PROGRAM Clamp_and_cut
VAR
	
	
	SawHome: BOOL; //Indexer is retracted to HOME switch
	SawTraversing: BOOL; // Saw is cycling through cutting
	SawDwellTimer: ton; // Dwell timer to wait for saw to spool up to speed
	SawExtended: BOOL; // Saw slide is fully extended
	ClampOpen: BOOL; // Saw clamp is open to receive part
	ClampClosed: BOOL; // Saw clamp is closed on to the part
	SawMotorRunning: BOOL; // Saw blade is spinning and motor not faulted
	CloseClampRequest: BOOL; // Logic bit to close saw clamp
	OpenClampRequest: BOOL; // Logic bit to open saw clamp
	SawDwellTimerElapsed: TIME; // Elapsed time of dwell timer
	SawDwellDoneBit: BOOL; // Dwell timer done bit
	StartSawRequest: BOOL; // Logic bit to start saw motor
	TraverseDwellTimer: ton; // Dwell timer to wait for traverse motor to spool up to speed
	TraverseDwellTimerElapsed: TIME; // Elapsed time of dwell timer
	TraverseDwellDoneBit: BOOL; // Dwell timer done bit
	DustCollectStartRequest: BOOL; // Logic bit to start dust collector
	
END_VAR
VAR // added by the converter: edge detectors and wires of the graphical bodies
    _rt1, _rt2, _rt3 : R_TRIG;
    _w1 : BOOL;
END_VAR

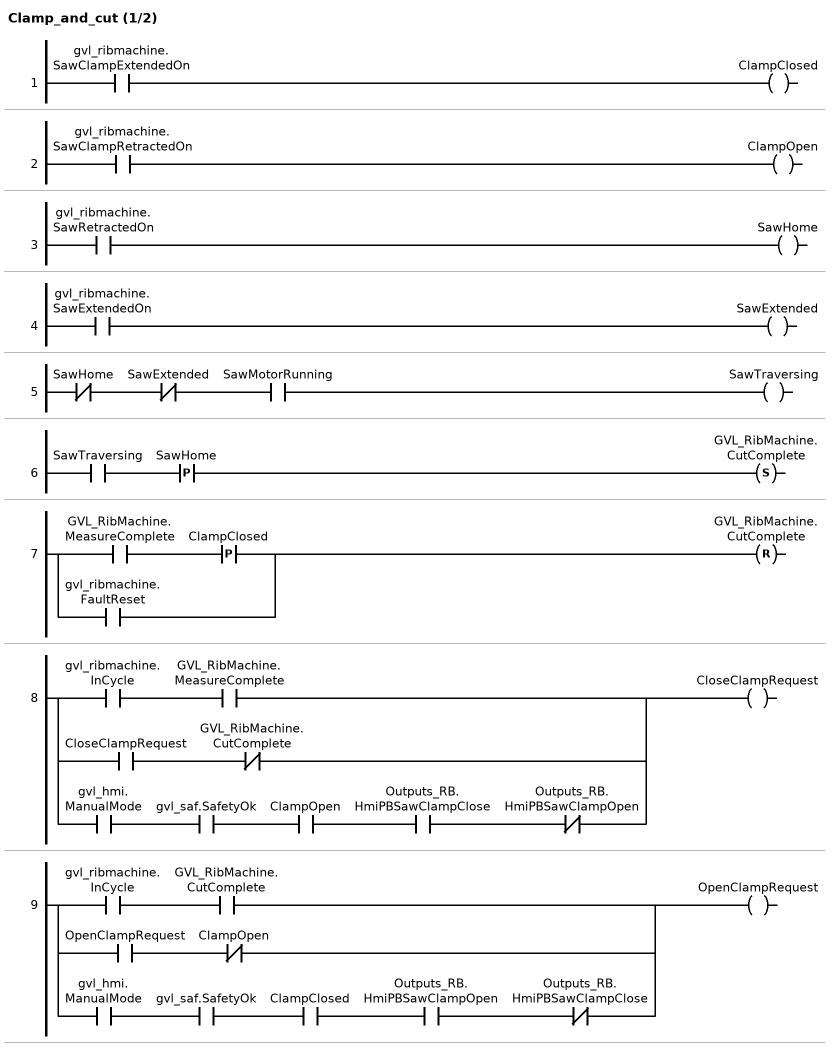
// NETWORK 1
ClampClosed := gvl_ribmachine.SawClampExtendedOn;

// NETWORK 2
ClampOpen := gvl_ribmachine.SawClampRetractedOn;

// NETWORK 3
SawHome := gvl_ribmachine.SawRetractedOn;

// NETWORK 4
SawExtended := gvl_ribmachine.SawExtendedOn;

// NETWORK 5
SawTraversing := NOT SawHome AND NOT SawExtended AND SawMotorRunning;

// NETWORK 6
_rt1(CLK := SawHome);
GVL_RibMachine.CutComplete S= SawTraversing AND _rt1.Q;

// NETWORK 7
_rt2(CLK := ClampClosed);
GVL_RibMachine.CutComplete R= GVL_RibMachine.MeasureComplete AND _rt2.Q OR gvl_ribmachine.FaultReset;

// NETWORK 8
CloseClampRequest := gvl_ribmachine.InCycle AND GVL_RibMachine.MeasureComplete OR CloseClampRequest AND NOT GVL_RibMachine.CutComplete OR gvl_hmi.ManualMode AND gvl_saf.SafetyOk AND ClampOpen AND Outputs_RB.HmiPBSawClampClose AND NOT Outputs_RB.HmiPBSawClampOpen;

// NETWORK 9
OpenClampRequest := gvl_ribmachine.InCycle AND GVL_RibMachine.CutComplete OR OpenClampRequest AND NOT ClampOpen OR gvl_hmi.ManualMode AND gvl_saf.SafetyOk AND ClampClosed AND Outputs_RB.HmiPBSawClampOpen AND NOT Outputs_RB.HmiPBSawClampClose;

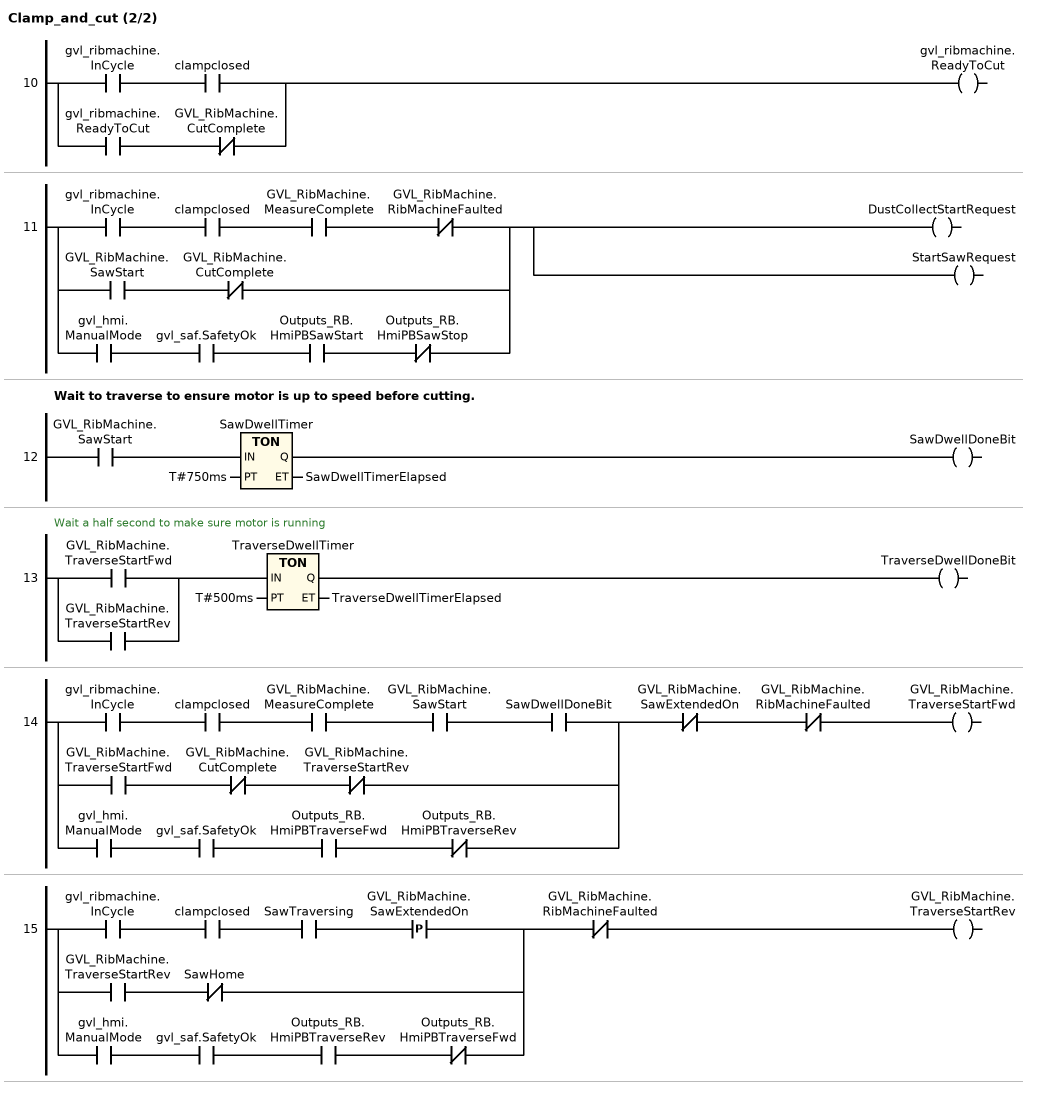
// NETWORK 10
gvl_ribmachine.ReadyToCut := gvl_ribmachine.InCycle AND clampclosed OR gvl_ribmachine.ReadyToCut AND NOT GVL_RibMachine.CutComplete;

// NETWORK 11
_w1 := gvl_ribmachine.InCycle AND clampclosed AND GVL_RibMachine.MeasureComplete AND NOT GVL_RibMachine.RibMachineFaulted OR GVL_RibMachine.SawStart AND NOT GVL_RibMachine.CutComplete OR gvl_hmi.ManualMode AND gvl_saf.SafetyOk AND Outputs_RB.HmiPBSawStart AND NOT Outputs_RB.HmiPBSawStop;
DustCollectStartRequest := _w1;
StartSawRequest := _w1;

// NETWORK 12: Wait to traverse to ensure motor is up to speed before cutting.
SawDwellTimer(IN := GVL_RibMachine.SawStart, PT := T#750ms, ET => SawDwellTimerElapsed); // TON
SawDwellDoneBit := SawDwellTimer.Q;

// NETWORK 13
// Wait a half second to make sure motor is running
TraverseDwellTimer(
    IN := GVL_RibMachine.TraverseStartFwd OR GVL_RibMachine.TraverseStartRev,
    PT := T#500ms,
    ET => TraverseDwellTimerElapsed); // TON
TraverseDwellDoneBit := TraverseDwellTimer.Q;

// NETWORK 14
GVL_RibMachine.TraverseStartFwd := (gvl_ribmachine.InCycle AND clampclosed AND GVL_RibMachine.MeasureComplete AND GVL_RibMachine.SawStart AND SawDwellDoneBit OR GVL_RibMachine.TraverseStartFwd AND NOT GVL_RibMachine.CutComplete AND NOT GVL_RibMachine.TraverseStartRev OR gvl_hmi.ManualMode AND gvl_saf.SafetyOk AND Outputs_RB.HmiPBTraverseFwd AND NOT Outputs_RB.HmiPBTraverseRev) AND NOT GVL_RibMachine.SawExtendedOn AND NOT GVL_RibMachine.RibMachineFaulted;

// NETWORK 15
_rt3(CLK := GVL_RibMachine.SawExtendedOn);
GVL_RibMachine.TraverseStartRev := (gvl_ribmachine.InCycle AND clampclosed AND SawTraversing AND _rt3.Q OR GVL_RibMachine.TraverseStartRev AND NOT SawHome OR gvl_hmi.ManualMode AND gvl_saf.SafetyOk AND Outputs_RB.HmiPBTraverseRev AND NOT Outputs_RB.HmiPBTraverseFwd) AND NOT GVL_RibMachine.RibMachineFaulted;

END_PROGRAM

(* stored: Version 1.1.0.1, ProductVersion 3.1.4024.12
   POU Clamp_and_cut: Id {b5b77416-dee0-4c77-a893-e09a1a73be42}, SpecialFunc None *)
